FUNCTION_BLOCK OrientStation EXTENDS MachineStation
VAR_INPUT
	rIO				: REFERENCE TO Orient_IO_typ;
	rStation		: REFERENCE TO Station;
	rBallSeatStn	: REFERENCE TO Station;
	rKickoutStn		: REFERENCE TO Station;
END_VAR
VAR_OUTPUT
END_VAR
VAR
	Payload	: Payload_typ;
END_VAR

(*IF rStation = 0 OR rIO = 0 THEN		HOW DO I CHECK FOR THIS???
	RETURN;
END_IF	*)

IF Enable THEN
	IF NOT _Enable THEN
		;
	END_IF

	CASE State OF
		STN_WAIT:
			IF Run AND rStation.MoverInPosition THEN
				State	:= STN_CHECKMOVER;
				Payload	:= rStation.CurrentMover.Payload;
			END_IF

		STN_CHECKMOVER:
			IF NOT Payload.Init THEN
				Payload.Init	:= TRUE;
			END_IF

			IF rIO.Inputs.BallPresent THEN
				// DO NOTHING FOR NOW
			ELSE
				rIO.Outputs.BallClampOpen	:= TRUE;
				State						:= STN_OPENBALLCLAMP;
			END_IF

		STN_OPENBALLCLAMP:
			IF rIO.Inputs.BallClampOpened THEN
				rIO.Outputs.BallClampOpen	:= FALSE;
				rIO.Outputs.LoadBall		:= TRUE;
				State						:= STN_PROCESS;
			END_IF

		STN_PROCESS:
			IF rIO.Inputs.BallLoadComplete THEN
				rIO.Outputs.LoadBall		:= FALSE;
				Payload.HasBall				:= TRUE;
				rIO.Outputs.BallClampClose	:= TRUE;
				State						:= STN_CLOSEBALLCLAMP;
			END_IF

		STN_CLOSEBALLCLAMP:
			IF rIO.Inputs.BallClampClosed THEN
				rIO.Outputs.BallClampClose	:= FALSE;
				State						:= STN_SEND;
			END_IF

		STN_SEND:
			rStation.CurrentMover.Payload	:= Payload;
			rStation.CurrentMover.MoveToStation(rBallSeatStn);
			rStation.UnregisterCurrent();
			State							:= STN_WAIT;
		
		STN_ERROR:
	
	END_CASE

ELSIF _Enable THEN
	;
END_IF

//Save Previous Values
_Enable	:= Enable;

METHOD Cyclic : BOOL
VAR_INPUT
END_VAR
END_METHOD

END_FUNCTION_BLOCK

(* stored: Version 1.1.0.1, ProductVersion 3.1.4024.12
   POU OrientStation: Id {37722a1a-8fe0-0ed5-3944-0550e379750d}, SpecialFunc None
   Method Cyclic: Id {a820a9db-2ef7-0ad2-29be-a32b40c3d2e1} *)
